FUNCTION_BLOCK E_CYCLE
  (* Standard: 61499-2 *)
  (* Version 10-12-2013, IECVM *)
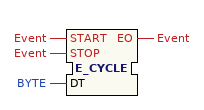
  EVENT_INPUT
    START;
    STOP;
  END_EVENT
  EVENT_OUTPUT
    EO;
  END_EVENT
  VAR_INPUT
    DT : BYTE;
  END_VAR
  EC_STATES
    START;
  END_STATES
END_FUNCTION_BLOCK
